// TwinCAT 3 PLC project GENE_PLC_Program
// ProgramVersion: 3.1.4022.1
// libraries:
//   Tc2_MC2, * (Beckhoff Automation GmbH)
//   Tc2_Standard, * (Beckhoff Automation GmbH)
//   Tc2_System, * (Beckhoff Automation GmbH)
//   Tc3_Module, * (Beckhoff Automation GmbH)
// project tree:
//   / PlcTask.TcTTO
//   POUs/P0_Start/ MAIN.TcPOU, P0_Start_Initialization.TcPOU
//   POUs/Variable/GVL_00_IO/ GVL_00_IO.TcGVL
//   POUs/Variable/GVL_01_Flag_Function/ GVL_01_Flag.TcGVL, GVL_01_Function.TcGVL, GVL_01_Shift.TcGVL, GVL_01_Station.TcGVL
//   POUs/Variable/GVL_02_Parameter/ GVL_02_Parameter_Common.TcGVL, GVL_02_Parameter_Output.TcGVL, GVL_02_Parameter_Servo_Motor_Robot.TcGVL, GVL_02_Parameter_Servo_Motor_Shelf_C.TcGVL, GVL_02_Parameter_Servo_Motor_Shelf_Z.TcGVL, GVL_02_Parameter_Servo_Motor_Shelf_Y.TcGVL, GVL_02_Parameter_Step_Motor_BOX_X.TcGVL, GVL_02_Parameter_Step_Motor_BOX_Y.TcGVL, GVL_02_Parameter_Step_Motor_Other.TcGVL
//   POUs/Variable/GVL_03_Delay/ GVL_03_Delay_Common.TcGVL, GVL_03_Delay_Output.TcGVL, GVL_03_Delay_Servo_Motor.TcGVL, GVL_03_Delay_Step_Motor.TcGVL
//   POUs/Variable/GVL_04_Auto/ GVL_04_Auto_All.TcGVL, GVL_04_Auto_Other.TcGVL, GVL_04_Auto_Servo_Motor.TcGVL, GVL_04_Auto_Step_Motor.TcGVL
//   POUs/Variable/GVL_05_Manual/ GVL_05_Manual_All.TcGVL, GVL_05_Manual_Servo_Motor_Robot.TcGVL, GVL_05_Manual_Servo_Motor_Shelf_C.TcGVL, GVL_05_Manual_Servo_Motor_Shelf_Y.TcGVL, GVL_05_Manual_Servo_Motor_Shelf_Z.TcGVL, GVL_05_Manual_Step_Motor_BOX_X.TcGVL, GVL_05_Manual_Step_Motor_BOX_Y.TcGVL, GVL_05_Manual_Step_Motor_Other.TcGVL, GVL_05_Manual_Test.TcGVL
//   POUs/Variable/GVL_06_Output/ GVL_06_Output_Other.TcGVL, GVL_06_Output_Servo_Motor_Robot.TcGVL, GVL_06_Output_Servo_Motor_Shelf_C.TcGVL, GVL_06_Output_Servo_Motor_Shelf_Y.TcGVL, GVL_06_Output_Servo_Motor_Shelf_Z.TcGVL, GVL_06_Output_Step_Motor.TcGVL
//   POUs/Variable/GVL_07_Alarm/ GVL_07_Alarm_Common.TcGVL, GVL_07_Alarm_Other.TcGVL, GVL_07_Alarm_Servo_Motor_Robot.TcGVL, GVL_07_Alarm_Servo_Motor_Shelf_C.TcGVL, GVL_07_Alarm_Servo_Motor_Shelf_Y.TcGVL, GVL_07_Alarm_Servo_Motor_Shelf_Z.TcGVL, GVL_07_Alarm_Step_Motor.TcGVL
// real-time tasks:
//   TASK PlcTask: cycle T#10ms, priority 20, ADS port 350
// motion (NC):
//   TASK NC-Task 1 SAF: cycle T#2ms, priority 4, ADS port 501
//   TASK NC-Task 1 SVB: cycle T#10ms, priority 8, ADS port 511
//   AXIS Axis 1 (id 1)
//     OtherSettings: AllowMotionCmdToSlave=true
//     encoder EncType=1
//     drive DrvType=5
//       Analog: ScaleFactorActTorque=0.1
//     controller CtrType=1
//       CtrPara: PriorControlFactor=1
//         Observer: BandWidth=20

CONFIGURATION GENE_PLC_Program
    RESOURCE PLC ON TwinCAT3
        TASK PlcTask(INTERVAL := T#10ms, PRIORITY := 20);
        PROGRAM MAIN WITH PlcTask : MAIN;
    END_RESOURCE
END_CONFIGURATION

// ---- POUs/Variable/GVL_00_IO/GVL_00_IO.TcGVL
{attribute 'qualified_only'}
VAR_GLOBAL
	//面板急停按钮
   Panel_EMG_Stop_Button                                 AT %IX4.0 :BOOL;
   //暂存区旋转门
   ZC_Step_Motor_Revolution_Door_Open_Sensor             AT %IX4.1 :BOOL;     
   ZC_Step_Motor_Revolution_Door_Close_Sensor            AT %IX4.2 :BOOL;
  //暂存区横向门 
   ZC_Step_Motor_Lateral_Door_Open_Sensor                AT %IX4.3 :BOOL;
   ZC_Step_Motor_Lateral_Door_Close_Sensor               AT %IX4.4 :BOOL;
   //暂存区升降机构
   ZC_Step_Motor_Elevator_Mechanism_Up_Sensor            AT %IX4.5 :BOOL;
   ZC_Step_Motor_Elevator_Mechanism_Down_Sensor          AT %IX4.6 :BOOL;
   //常温区传送机构
   CW_Step_Motor_Transport_In_Sensor                     AT %IX4.7 :BOOL;
   CW_Step_Motor_Transport_Out_Sensor                    AT %IX4.8 :BOOL;
   //常温区保温门
   CW_Step_Motor_Door_Up_Sensor                          AT %IX4.9 :BOOL;
   CW_Step_Motor_Door_Down_Sensor                        AT %IX4.10 :BOOL;
   CW_Step_Motor_Door_Forward_Sensor                     AT %IX4.11 :BOOL;
   CW_Step_Motor_Door_Backward_Sensor                    AT %IX4.12 :BOOL;
   //常温区机器人升降伺服电机
   CW_Servo_Motor_Robot_Up_Limit_Sensor                  AT %IX5.0  :BOOL;
   CW_Servo_Motor_Robot_Down_Limit_Sensor                AT %IX5.1  :BOOL;
   CW_Servo_Motor_Robot_Home_Sensor                      AT %IX5.2  :BOOL; 
   
   //常温区料架前后伺服电机
   CW_Servo_Motor_Shelf_Y_Forward_Limit_Sensor             AT %IX6.0  :BOOL;
   CW_Servo_Motor_Shelf_Y_Backward_Limit_Sensor            AT %IX6.1  :BOOL;
   CW_Servo_Motor_Shelf_Home_Sensor                        AT %IX6.2  :BOOL;
   //常温区料架上下伺服电机
   CW_Servo_Motor_Shelf_Z_Up_Limit_Sensor                  AT %IX7.0  :BOOL;
   CW_Servo_Motor_Shelf_Z_Down_Limit_Sensor                AT %IX7.1  :BOOL;
   CW_Servo_Motor_Shelf_Z_Home_Sensor                      AT %IX7.2  :BOOL;
    //常温区料架旋转伺服电机
   CW_Servo_Motor_Shelf_C_Home_Sensor                      AT %IX7.3  :BOOL;
   //常温区卡料架步进电机
   CW_Step_Motor_Shelf_Escapement_Open_Sensor              AT %IX7.4  :BOOL;
   CW_Step_Motor_Shelf_Escapement_Close_Sensor             AT %IX7.5  :BOOL;
   //常温区机器人上是否有夹具感应
   CW_Is_Gripper_On_Robot_Sensor                           AT %IX7.6  :BOOL;
   //常温区夹爪1是否在夹爪座上
   CW_Is_Gripper1_On_Seat_Sensor                           AT %IX7.7  :BOOL;
   //常温区夹爪2是否在夹爪座上
   CW_Is_Gripper2_On_Seat_Sensor                           AT %IX7.8  :BOOL;
   //操作区取盒子步进电机
   CZ_Step_Motor_Box_X_Left_Sensor                         AT %IX7.9  :BOOL;
   CZ_Step_Motor_Box_X_Right_Sensor                        AT %IX8.0  :BOOL;
   CZ_Step_Motor_Box_X_Home_Sensor                         AT %IX8.1  :BOOL;
   //操作区盒子定位步进电机
   CZ_Step_Motor_Box_Y_Forward_Sensor                      AT %IX8.2  :BOOL;
   CZ_Step_Motor_Box_Y_Backward_Sensor                     AT %IX8.3  :BOOL;
   CZ_Step_Motor_Box_Y_Home_Sensor                         AT %IX8.4  :BOOL;
   
    
   
END_VAR

// ---- POUs/Variable/GVL_01_Flag_Function/GVL_01_Flag.TcGVL
{attribute 'qualified_only'}
VAR_GLOBAL
END_VAR

// ---- POUs/Variable/GVL_01_Flag_Function/GVL_01_Function.TcGVL
{attribute 'qualified_only'}
VAR_GLOBAL
END_VAR

// ---- POUs/Variable/GVL_01_Flag_Function/GVL_01_Shift.TcGVL
{attribute 'qualified_only'}
VAR_GLOBAL
END_VAR

// ---- POUs/Variable/GVL_01_Flag_Function/GVL_01_Station.TcGVL
{attribute 'qualified_only'}
VAR_GLOBAL
END_VAR

// ---- POUs/Variable/GVL_02_Parameter/GVL_02_Parameter_Common.TcGVL
{attribute 'qualified_only'}
VAR_GLOBAL
END_VAR

// ---- POUs/Variable/GVL_02_Parameter/GVL_02_Parameter_Output.TcGVL
{attribute 'qualified_only'}
VAR_GLOBAL
END_VAR

// ---- POUs/Variable/GVL_02_Parameter/GVL_02_Parameter_Servo_Motor_Robot.TcGVL
{attribute 'qualified_only'}
VAR_GLOBAL
END_VAR

// ---- POUs/Variable/GVL_02_Parameter/GVL_02_Parameter_Servo_Motor_Shelf_C.TcGVL
{attribute 'qualified_only'}
VAR_GLOBAL
END_VAR

// ---- POUs/Variable/GVL_02_Parameter/GVL_02_Parameter_Servo_Motor_Shelf_Z.TcGVL
{attribute 'qualified_only'}
VAR_GLOBAL
END_VAR

// ---- POUs/Variable/GVL_02_Parameter/GVL_02_Parameter_Servo_Motor_Shelf_Y.TcGVL
{attribute 'qualified_only'}
VAR_GLOBAL
END_VAR

// ---- POUs/Variable/GVL_02_Parameter/GVL_02_Parameter_Step_Motor_BOX_X.TcGVL
{attribute 'qualified_only'}
VAR_GLOBAL
END_VAR

// ---- POUs/Variable/GVL_02_Parameter/GVL_02_Parameter_Step_Motor_BOX_Y.TcGVL
{attribute 'qualified_only'}
VAR_GLOBAL
END_VAR

// ---- POUs/Variable/GVL_02_Parameter/GVL_02_Parameter_Step_Motor_Other.TcGVL
{attribute 'qualified_only'}
VAR_GLOBAL
END_VAR

// ---- POUs/Variable/GVL_03_Delay/GVL_03_Delay_Common.TcGVL
{attribute 'qualified_only'}
VAR_GLOBAL
END_VAR

// ---- POUs/Variable/GVL_03_Delay/GVL_03_Delay_Output.TcGVL
{attribute 'qualified_only'}
VAR_GLOBAL
END_VAR

// ---- POUs/Variable/GVL_03_Delay/GVL_03_Delay_Servo_Motor.TcGVL
{attribute 'qualified_only'}
VAR_GLOBAL
END_VAR

// ---- POUs/Variable/GVL_03_Delay/GVL_03_Delay_Step_Motor.TcGVL
{attribute 'qualified_only'}
VAR_GLOBAL
END_VAR

// ---- POUs/Variable/GVL_04_Auto/GVL_04_Auto_All.TcGVL
{attribute 'qualified_only'}
VAR_GLOBAL
END_VAR

// ---- POUs/Variable/GVL_04_Auto/GVL_04_Auto_Other.TcGVL
{attribute 'qualified_only'}
VAR_GLOBAL
END_VAR

// ---- POUs/Variable/GVL_04_Auto/GVL_04_Auto_Servo_Motor.TcGVL
{attribute 'qualified_only'}
VAR_GLOBAL
END_VAR

// ---- POUs/Variable/GVL_04_Auto/GVL_04_Auto_Step_Motor.TcGVL
{attribute 'qualified_only'}
VAR_GLOBAL
END_VAR

// ---- POUs/Variable/GVL_05_Manual/GVL_05_Manual_All.TcGVL
{attribute 'qualified_only'}
VAR_GLOBAL
END_VAR

// ---- POUs/Variable/GVL_05_Manual/GVL_05_Manual_Servo_Motor_Robot.TcGVL
{attribute 'qualified_only'}
VAR_GLOBAL
END_VAR

// ---- POUs/Variable/GVL_05_Manual/GVL_05_Manual_Servo_Motor_Shelf_C.TcGVL
{attribute 'qualified_only'}
VAR_GLOBAL
END_VAR

// ---- POUs/Variable/GVL_05_Manual/GVL_05_Manual_Servo_Motor_Shelf_Y.TcGVL
{attribute 'qualified_only'}
VAR_GLOBAL
END_VAR

// ---- POUs/Variable/GVL_05_Manual/GVL_05_Manual_Servo_Motor_Shelf_Z.TcGVL
{attribute 'qualified_only'}
VAR_GLOBAL
END_VAR

// ---- POUs/Variable/GVL_05_Manual/GVL_05_Manual_Step_Motor_BOX_X.TcGVL
{attribute 'qualified_only'}
VAR_GLOBAL
END_VAR

// ---- POUs/Variable/GVL_05_Manual/GVL_05_Manual_Step_Motor_BOX_Y.TcGVL
{attribute 'qualified_only'}
VAR_GLOBAL
END_VAR

// ---- POUs/Variable/GVL_05_Manual/GVL_05_Manual_Step_Motor_Other.TcGVL
{attribute 'qualified_only'}
VAR_GLOBAL
END_VAR

// ---- POUs/Variable/GVL_05_Manual/GVL_05_Manual_Test.TcGVL
{attribute 'qualified_only'}
VAR_GLOBAL
END_VAR

// ---- POUs/Variable/GVL_06_Output/GVL_06_Output_Other.TcGVL
{attribute 'qualified_only'}
VAR_GLOBAL
END_VAR

// ---- POUs/Variable/GVL_06_Output/GVL_06_Output_Servo_Motor_Robot.TcGVL
{attribute 'qualified_only'}
VAR_GLOBAL
END_VAR

// ---- POUs/Variable/GVL_06_Output/GVL_06_Output_Servo_Motor_Shelf_C.TcGVL
{attribute 'qualified_only'}
VAR_GLOBAL
END_VAR

// ---- POUs/Variable/GVL_06_Output/GVL_06_Output_Servo_Motor_Shelf_Y.TcGVL
{attribute 'qualified_only'}
VAR_GLOBAL
END_VAR

// ---- POUs/Variable/GVL_06_Output/GVL_06_Output_Servo_Motor_Shelf_Z.TcGVL
{attribute 'qualified_only'}
VAR_GLOBAL
END_VAR

// ---- POUs/Variable/GVL_06_Output/GVL_06_Output_Step_Motor.TcGVL
{attribute 'qualified_only'}
VAR_GLOBAL
	
    //暂存区旋转门
    ZC_Step_Motor_Revolution_Door_Direction           AT %QX4.0 :BOOL;
    ZC_Step_Motor_Revolution_Door_Switch              AT %QX4.1 :BOOL;
	//暂存区横移门
    ZC_Step_Motor_Lateral_Door_Direction              AT %QX4.2 :BOOL;
	ZC_Step_Motor_Lateral_Door_Switch                 AT %QX4.3 :BOOL;
	//暂存区升降机构
	ZC_Step_Motor_Elevator_Mechanism_Direction        AT %QX4.4 :BOOL;	
    ZC_Step_Motor_Elevator_Mechanism_Switch           AT %QX4.5 :BOOL;
	//常温区盒子传送电机
	CW_Step_Motor_Transport_Direction                 AT %QX5.0 :BOOL;
    CW_Step_Motor_Transport_Switch                    AT %QX5.1 :BOOL;
	CW_Step_Motor_Transport_Inch                      AT %QX5.2 :BOOL;
    //常温区门上下步进电机
    CW_Step_Motor_Door_UpDown_Direction               AT %QX5.3 :BOOL;
    CW_Step_Motor_Door_UpDown_Switch                  AT %QX5.4 :BOOL;
	//常温区门前后电机
	CW_Step_Motor_Door_FB_Direction                   AT %QX5.5 :BOOL;
	CW_Step_Motor_Door_FB_Switch                      AT %QX5.6 :BOOL;
	//常温区卡料架电机
	CW_Step_Motor_Shelf_Escapement_Direction          AT %QX5.7 :BOOL;
	CW_Step_Motor_Shelf_Escapement_Switch             AT %QX5.8 :BOOL;
	

END_VAR

// ---- POUs/Variable/GVL_07_Alarm/GVL_07_Alarm_Common.TcGVL
{attribute 'qualified_only'}
VAR_GLOBAL
END_VAR

// ---- POUs/Variable/GVL_07_Alarm/GVL_07_Alarm_Other.TcGVL
{attribute 'qualified_only'}
VAR_GLOBAL
END_VAR

// ---- POUs/Variable/GVL_07_Alarm/GVL_07_Alarm_Servo_Motor_Robot.TcGVL
{attribute 'qualified_only'}
VAR_GLOBAL
END_VAR

// ---- POUs/Variable/GVL_07_Alarm/GVL_07_Alarm_Servo_Motor_Shelf_C.TcGVL
{attribute 'qualified_only'}
VAR_GLOBAL
END_VAR

// ---- POUs/Variable/GVL_07_Alarm/GVL_07_Alarm_Servo_Motor_Shelf_Y.TcGVL
{attribute 'qualified_only'}
VAR_GLOBAL
END_VAR

// ---- POUs/Variable/GVL_07_Alarm/GVL_07_Alarm_Servo_Motor_Shelf_Z.TcGVL
{attribute 'qualified_only'}
VAR_GLOBAL
END_VAR

// ---- POUs/Variable/GVL_07_Alarm/GVL_07_Alarm_Step_Motor.TcGVL
{attribute 'qualified_only'}
VAR_GLOBAL
END_VAR

// ---- POUs/P0_Start/MAIN.TcPOU
PROGRAM MAIN
VAR
	
	B_out :BOOL;
	B_in  :BOOL;

END_VAR

P0_Start_Initialization();
B_out := B_in;

END_PROGRAM

// ---- POUs/P0_Start/P0_Start_Initialization.TcPOU
PROGRAM P0_Start_Initialization
VAR
END_VAR

END_PROGRAM
